PROGRAM Alias
VAR
	i : INT := 0;
END_VAR

//R1 : MCP**  
	//DI
	
	MCP_IO.EStopPB_NotPressed					:= Input.R1_01_00;  //NC - 
	MCP_IO.DoorSWclose							:= Input.R1_01_01;  
	MCP_IO.ShortContactClose					:= Input.R1_01_02; 
	MCP_IO.UnshortContactClose					:= Input.R1_01_03; 
	//MCP_IO.MachineGNDrlyOpen					:= Input.R1_01_04; // machine ground lifted (opto board)	
	//MCP_IO.CloseAllChargeRlyCommand				:= Input.R1_01_05; // command from screen room (opto) - Slim only
	//MCP_IO.OpenAllDumpRelayCommand				:= Input.R1_01_06; // command from screen room (opto) - slim only
	
	
	//INPUT
	//DI
	MCP_IO.Charger[1].inhibited					:= NOT Input.R1_02_00; //TDK802 1 NC for all feedback esaigeean
	MCP_IO.Charger[1].EndOfCharge				:= NOT Input.R1_02_01; //TDK802 1
	MCP_IO.Charger[1].HV_isON					:= NOT Input.R1_02_02; //TDK802 1
	MCP_IO.Charger[1].SummaryFaulted			:= NOT Input.R1_02_03; //TDK802 1
	//MCP_IO.Charger[1].OverTemp					:= Input.R1_02_03; //TDK802 1
	//MCP_IO.Charger[1].InterlockOpen				:= Input.R1_02_04; //TDK802 1
	//MCP_IO.Charger[1].LoadFaulted				:= Input.R1_02_05; //TDK802 1
	
	LCP1_IO.Segment[1].Module[1].ChargeRly_close := Input.R1_02_04;
	LCP1_IO.Segment[1].Module[1].DumpRly_open	 := NOT Input.R1_02_05;
	
	//EL3068 - AI
	MCP_IO.Charger[1].voltageFeedback_raw		:= Input.R1_04_00;
	MCP_IO.Charger[1].currentFeedback_raw		:= Input.R1_04_01;
	//OUTPUT
	//DQ
	Output.R1_03_00								:= MCP_IO.Charger[1].inhibit;
	Output.R1_03_01								:= MCP_IO.Charger[1].HV_ON;
	Output.R1_03_02								:= LCP1_IO.Segment[1].Module[1].CloseChargeRly;
	Output.R1_03_03								:= LCP1_IO.Segment[1].Module[1].OpenDumpRly;
	Output.R1_03_04								:= LCP1_IO.Segment[1].Module[1].Fire;
	Output.R1_03_05								:= LCP1_IO.Segment[1].Module[1].TriggerScope;
	Output.R1_03_06								:= MCP_IO.EnergizeACKontactor;
	Output.R1_03_07								:= LCP1_IO.Segment[1].Module[1].ModuleCharged;
	//AQ
	Output.R1_05_00								:= MCP_IO.Charger[1].voltageSP_raw;
	
	//Cap voltage monitor feedback is at VoltMonitor
	VoltMonitor_DB.CapRaw[0] 					:= Input.B170357_CapRaw[0]; 
	FOR i := 1 TO 24 BY 1 DO 
		VoltMonitor_DB.CapRaw[i] 					:= Input.B170357_CapRaw[i]; 
	END_FOR
	
IF i > 24 THEN
	i := 0;
END_IF
	
//*************************************************************************************************************

END_PROGRAM

(* stored: Version 1.1.0.1, ProductVersion 3.1.4024.11
   POU Alias: Id {ebc75665-f0df-4b03-b4d1-48515468f179}, SpecialFunc None *)
